Fanuc KAREL source: wcntshortmo.kl

PROGRAM wcntshortmo
%NOLOCKGROUP
VAR
  p : POSITION
  q : POSITION
  i : INTEGER
  r : REAL
BEGIN
  WITH $CNT_SHORTMO = TRUE MOVE TO p
END wcntshortmo
